{attribute 'GeneratedUsingTerminal: EPP5001-0002-0016'}
{attribute addProperty BoxType "EPP5001-0002-0016"}
{attribute addProperty Id "EtcSlaveTerminalBaseSSI_InputsAT %I*SSI_Inputs_0E3D8E3310WcStateAT %I*WcState_9091E0EB2InfoDataAT %I*InfoData_32EB74EA10"}
{attribute addProperty CRC "151481710"}
{attribute addProperty Size "22"}
TYPE EPP5001_09076D6E EXTENDS EtcSlaveTerminalBase :
STRUCT
	{attribute addProperty Name "SSI_Inputs"}
	SSI_Inputs : SSI_Inputs_0E3D8E33;
	{attribute addProperty Name "WcState"}
	WcState : WcState_9091E0EB;
	{attribute addProperty Name "InfoData"}
	InfoData : InfoData_32EB74EA;
END_STRUCT
END_TYPE

(* stored: Version 1.2.0.0, ProductVersion 3.1.4024.9
   DUT EPP5001_09076D6E: Id {90fb238d-c861-434f-b339-ae6551a2c076} *)
